// TIA Portal V15.1 export
// export: Created 2020-06-12T07:35:54.4755859Z, ExportSetting None, DisplayName Totally Integrated Automation Portal, DisplayVersion V15.1, DisplayName TIA Portal Openness, DisplayVersion V15.1, DisplayName STEP 7 Professional, DisplayVersion V15.1, DisplayName STEP 7 Safety, DisplayVersion V15.1, DisplayName WinCC Advanced, DisplayVersion V15.1
FUNCTION "Desk_call" : Void   // FC163, FBD
TITLE = Desks indication
{ S7_Optimized_Access := 'TRUE' }
// stored: SetENOAutomatically False
BEGIN

REGION Network 1
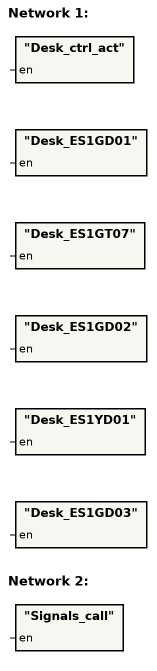
   "Desk_ctrl_act"();
   "Desk_ES1GD01"();
   "Desk_ES1GT07"();
   "Desk_ES1GD02"();
   "Desk_ES1YD01"();
   "Desk_ES1GD03"();
END_REGION

REGION Network 2
   "Signals_call"();
END_REGION
END_FUNCTION
